ABB RobotStudio station: PiecePicking_20230616-110847.rsstn

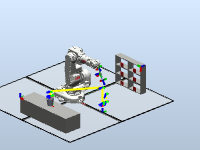
Station PiecePicking (saved by RobotStudio 6.8.8307.1040)
Controller System1
  mechanical unit ROB_1: IRB140_6_81_C_03, 6 joints, base frame (0, 0, 0) mm
Layout (positions relative to the parent item):
  - IRB140_6_81_C_03 [mechanism, from Robots\IRB140_6_81_C_G_03.rslib] at (0, 0, 0) mm; joint values [0, 0, 0, 0, 0.5236, 0] (rad or m)
  - Banda [part, from Libraries\Banda.rslib] at (-200, -850, 0) mm, rotated rx 90 ry 0 rz 90 deg
  - Balde [part, from Libraries\Balde.rslib] at (275, -710, 235) mm, rotated rx 90 ry 0 rz 90 deg
  - EstanteriaA  [part, from Libraries\EstanteriaA .rslib] at (0, 900, 0) mm, rotated rx 90 ry 0 rz 0 deg
  - Positioner_Balde [smart component, from Components\Positioner.rslib]
      properties: Object=Balde; Position=[0.275 -0.71 0.235]; Orientation=[1.5707963267949 0 1.5707963267949]; Reference=Global; ReferenceObject=(none)
  - Attacher_Balde [smart component, from Components\Attacher.rslib]
      properties: Parent=PF_Robotica; Flange=0; Child=Balde; Mount=false; Offset=[0 0 0]; Orientation=[0 0 0]
  - Detacher_Balde [smart component, from Components\Detacher.rslib]
      properties: Child=Balde; KeepPosition=true
  - PF_Robotica [mechanism, from Libraries\PF_Robotica.rslib] at (506.29, 0, 679.5) mm, rotated rx 180 ry 60 rz 180 deg
  - Pieza1 [smart component, from Libraries\Pieza1.rslib] at (-245.55, 1050.01, 0) mm
      connections:
        Pieza1.Pos_Pieza1 -> Positioner.Execute
        Pieza1.Attach_Pieza -> Attacher.Execute
        Pieza1.Detach_pieza -> Detacher.Execute
    - Positioner [smart component, from Components\Positioner.rslib] at (88.58, 803, 328) mm, rotated rx -90 ry 0 rz 0 deg
        properties: Object=PiezaTest_1; Position=[0.39675 0.803 0.328]; Orientation=[-1.5707963267949 0 0]; Reference=Global; ReferenceObject=(none)
    - PiezaTest_1 [part, from Libraries\Pieza1.rslib] at (642.3, -247.01, 328) mm, rotated rx -90 ry 0 rz 0 deg
    - Attacher [smart component, from Components\Attacher.rslib]
        properties: Parent=PF_Robotica; Flange=1; Child=PiezaTest_1; Mount=false; Offset=[0 0 0]; Orientation=[0 0 0]
    - Detacher [smart component, from Components\Detacher.rslib]
        properties: Child=PiezaTest_1; KeepPosition=true
  - Pieza2 [smart component, from Libraries\Pieza1.rslib] at (-251.26, 1022.75, 0) mm
      connections:
        Pieza2.Pos_Pieza1 -> Positioner.Execute
        Pieza2.Attach_Pieza -> Attacher.Execute
        Pieza2.Detach_pieza -> Detacher.Execute
    - Positioner [smart component, from Components\Positioner.rslib] at (88.58, 803, 328) mm, rotated rx -90 ry 0 rz 0 deg
        properties: Object=PiezaTest_1; Position=[0.13625 0.803 0.328]; Orientation=[-1.5707963267949 0 0]; Reference=Global; ReferenceObject=(none)
    - PiezaTest_1 [part, from Libraries\Pieza1.rslib] at (387.51, -219.75, 328) mm, rotated rx -90 ry 0 rz 0 deg
    - Attacher [smart component, from Components\Attacher.rslib]
        properties: Parent=PF_Robotica; Flange=1; Child=PiezaTest_1; Mount=false; Offset=[0 0 0]; Orientation=[0 0 0]
    - Detacher [smart component, from Components\Detacher.rslib]
        properties: Child=PiezaTest_1; KeepPosition=true
  - Pieza3 [smart component, from Libraries\Pieza1.rslib] at (-251.26, 1022.75, 0) mm
      connections:
        Pieza3.Pos_Pieza1 -> Positioner.Execute
        Pieza3.Attach_Pieza -> Attacher.Execute
        Pieza3.Detach_pieza -> Detacher.Execute
    - Positioner [smart component, from Components\Positioner.rslib] at (88.58, 803, 328) mm, rotated rx -90 ry 0 rz 0 deg
        properties: Object=PiezaTest_1; Position=[0.13625 0.803 0.189]; Orientation=[-1.5707963267949 0 0]; Reference=Global; ReferenceObject=(none)
    - PiezaTest_1 [part, from Libraries\Pieza1.rslib] at (387.51, -219.75, 189) mm, rotated rx -90 ry 0 rz 0 deg
    - Attacher [smart component, from Components\Attacher.rslib]
        properties: Parent=PF_Robotica; Flange=1; Child=PiezaTest_1; Mount=false; Offset=[0 0 0]; Orientation=[0 0 0]
    - Detacher [smart component, from Components\Detacher.rslib]
        properties: Child=PiezaTest_1; KeepPosition=true
  - Pieza4 [smart component, from Libraries\Pieza1.rslib] at (-251.26, 1022.75, 0) mm
      connections:
        Pieza4.Pos_Pieza1 -> Positioner.Execute
        Pieza4.Attach_Pieza -> Attacher.Execute
        Pieza4.Detach_pieza -> Detacher.Execute
    - Positioner [smart component, from Components\Positioner.rslib] at (88.58, 803, 328) mm, rotated rx -90 ry 0 rz 0 deg
        properties: Object=PiezaTest_1; Position=[0.39675 0.803 0.189]; Orientation=[-1.5707963267949 0 0]; Reference=Global; ReferenceObject=(none)
    - PiezaTest_1 [part, from Libraries\Pieza1.rslib] at (648.01, -219.75, 189) mm, rotated rx -90 ry 0 rz 0 deg
    - Attacher [smart component, from Components\Attacher.rslib]
        properties: Parent=PF_Robotica; Flange=1; Child=PiezaTest_1; Mount=false; Offset=[0 0 0]; Orientation=[0 0 0]
    - Detacher [smart component, from Components\Detacher.rslib]
        properties: Child=PiezaTest_1; KeepPosition=true
  - Pieza5 [smart component, from Libraries\Pieza1.rslib] at (-251.26, 1022.75, 0) mm
      connections:
        Pieza5.Pos_Pieza1 -> Positioner.Execute
        Pieza5.Attach_Pieza -> Attacher.Execute
        Pieza5.Detach_pieza -> Detacher.Execute
    - Positioner [smart component, from Components\Positioner.rslib] at (88.58, 803, 328) mm, rotated rx -90 ry 0 rz 0 deg
        properties: Object=PiezaTest_1; Position=[0.13625 0.803 0.042]; Orientation=[-1.5707963267949 0 0]; Reference=Global; ReferenceObject=(none)
    - PiezaTest_1 [part, from Libraries\Pieza1.rslib] at (387.51, -219.75, 42) mm, rotated rx -90 ry 0 rz 0 deg
    - Attacher [smart component, from Components\Attacher.rslib]
        properties: Parent=PF_Robotica; Flange=1; Child=PiezaTest_1; Mount=false; Offset=[0 0 0]; Orientation=[0 0 0]
    - Detacher [smart component, from Components\Detacher.rslib]
        properties: Child=PiezaTest_1; KeepPosition=true
  - Pieza6 [smart component, from Libraries\Pieza1.rslib] at (-251.26, 1022.75, 0) mm
      connections:
        Pieza6.Pos_Pieza1 -> Positioner.Execute
        Pieza6.Attach_Pieza -> Attacher.Execute
        Pieza6.Detach_pieza -> Detacher.Execute
    - Positioner [smart component, from Components\Positioner.rslib] at (88.58, 803, 328) mm, rotated rx -90 ry 0 rz 0 deg
        properties: Object=PiezaTest_1; Position=[0.39675 0.803 0.042]; Orientation=[-1.5707963267949 0 0]; Reference=Global; ReferenceObject=(none)
    - PiezaTest_1 [part, from Libraries\Pieza1.rslib] at (648.01, -219.75, 42) mm, rotated rx -90 ry 0 rz 0 deg
    - Attacher [smart component, from Components\Attacher.rslib]
        properties: Parent=PF_Robotica; Flange=1; Child=PiezaTest_1; Mount=false; Offset=[0 0 0]; Orientation=[0 0 0]
    - Detacher [smart component, from Components\Detacher.rslib]
        properties: Child=PiezaTest_1; KeepPosition=true
Attachment: PF_Robotica is attached to IRB140_6_81_C_03 / Link6
Attachment: Workobject_Est is attached to EstanteriaA 
Attachment: Workobject_1 is attached to Banda
Station signals: DI Balde_positioner, DI Pos_Pieza1, DI Pos_Pieza2, DI Pos_Pieza3, DI Pos_Pieza4, DI Pos_Pieza5, DI Pos_Pieza6, DI Pos_Piezas, DO DO_01, DO DO_02
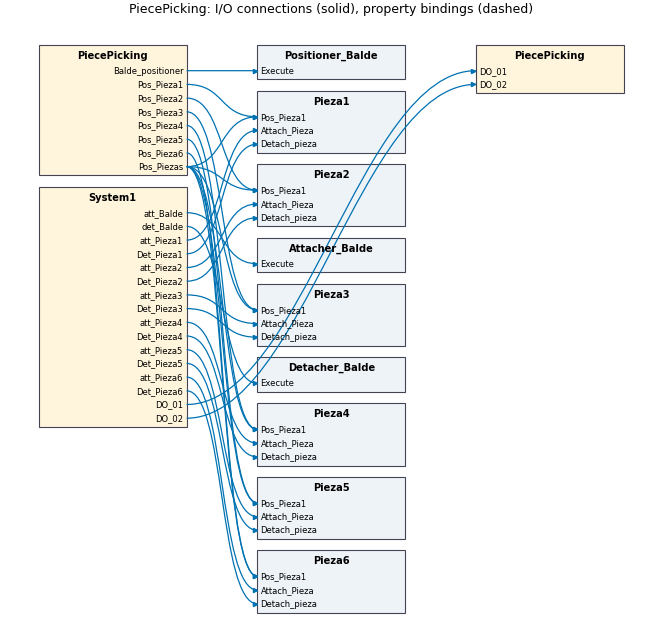
Station logic (signal -> signal, property => property):
  PiecePicking.Balde_positioner -> Positioner_Balde.Execute
  System1.att_Balde -> Attacher_Balde.Execute
  System1.det_Balde -> Detacher_Balde.Execute
  PiecePicking.Pos_Pieza1 -> Pieza1.Pos_Pieza1
  PiecePicking.Pos_Pieza2 -> Pieza2.Pos_Pieza1
  System1.att_Pieza1 -> Pieza1.Attach_Pieza
  System1.Det_Pieza1 -> Pieza1.Detach_pieza
  System1.att_Pieza2 -> Pieza2.Attach_Pieza
  System1.Det_Pieza2 -> Pieza2.Detach_pieza
  PiecePicking.Pos_Pieza3 -> Pieza3.Pos_Pieza1
  PiecePicking.Pos_Pieza4 -> Pieza4.Pos_Pieza1
  PiecePicking.Pos_Pieza5 -> Pieza5.Pos_Pieza1
  PiecePicking.Pos_Pieza6 -> Pieza6.Pos_Pieza1
  PiecePicking.Pos_Piezas -> Pieza6.Pos_Pieza1
  PiecePicking.Pos_Piezas -> Pieza5.Pos_Pieza1
  PiecePicking.Pos_Piezas -> Pieza4.Pos_Pieza1
  PiecePicking.Pos_Piezas -> Pieza3.Pos_Pieza1
  PiecePicking.Pos_Piezas -> Pieza2.Pos_Pieza1
  PiecePicking.Pos_Piezas -> Pieza1.Pos_Pieza1
  System1.att_Pieza3 -> Pieza3.Attach_Pieza
  System1.Det_Pieza3 -> Pieza3.Detach_pieza
  System1.att_Pieza4 -> Pieza4.Attach_Pieza
  System1.Det_Pieza4 -> Pieza4.Detach_pieza
  System1.att_Pieza5 -> Pieza5.Attach_Pieza
  System1.Det_Pieza5 -> Pieza5.Detach_pieza
  System1.att_Pieza6 -> Pieza6.Attach_Pieza
  System1.Det_Pieza6 -> Pieza6.Detach_pieza
  System1.DO_01 -> PiecePicking.DO_01
  System1.DO_02 -> PiecePicking.DO_02
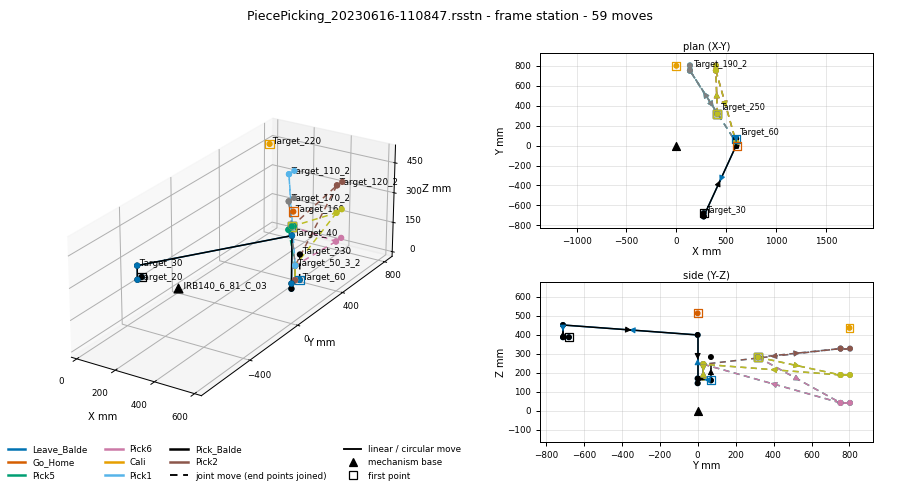
[picture p0: tool path of PiecePicking_20230616-110847.rsstn in frame station, 59 of 59 moves have a stored position in this frame; points joined in program order, loops and branches not executed]
Targets, tools, work objects and paths stored in the station, written as RAPID:
! task T_ROB1
MODULE CalibData
  TASK PERS wobjdata Workobject_1:=[FALSE,TRUE,"",[[-200,-850,230],[1,0,0,0]],[[475,140,0],[1,0,0,0]]];
  PERS tooldata TD_Hook:=[TRUE,[[68.38,0,60],[0.707106781,0.707106781,0,0]],[0.2,[28.798,-0.092,56.062],[1,0,0,0],0,0,0]];
  PERS tooldata TD_SuctionPad:=[TRUE,[[93.75,0,168.37],[0.970295726,0,0.241921896,0]],[0.2,[28.798,-0.092,56.062],[1,0,0,0],0,0,0]];
  TASK PERS wobjdata Workobject_Balde_Piso:=[FALSE,TRUE,"",[[600,0,0],[1,0,0,0]],[[0,0,0],[1,0,0,0]]];
  TASK PERS wobjdata Workobject_Est:=[FALSE,TRUE,"",[[533,800,437],[0.5,-0.5,0.5,0.5]],[[0,0,0],[1,0,0,0]]];
ENDMODULE

! task T_ROB1
MODULE Module1
  CONST robtarget Target_20:=[[-0.54180672,0.235098408,157.927793799],[0.499363871,0.499363893,0.500635292,-0.500635328],[-1,1,-2,0],[9E+09,9E+09,9E+09,9E+09,9E+09,9E+09]];
  CONST robtarget Target_10:=[[-0.541791285,31.542690631,157.927772118],[0.338220375,0.61994805,0.62152642,-0.339081557],[-1,1,-1,0],[9E+09,9E+09,9E+09,9E+09,9E+09,9E+09]];
  CONST robtarget Target_30:=[[-0.541814528,0.23509908,222.389598203],[0.499363884,0.49936382,0.500635317,-0.500635363],[-1,1,-2,0],[9E+09,9E+09,9E+09,9E+09,9E+09,9E+09]];
  CONST robtarget Target_40:=[[0,0,400],[0.499363884,0.49936382,0.500635317,-0.500635363],[0,1,-3,0],[9E+09,9E+09,9E+09,9E+09,9E+09,9E+09]];
  CONST robtarget Target_50:=[[-0.038127492,-0.000030739,145.519742619],[0.499363836,0.499363825,0.500635306,-0.500635416],[-1,2,-3,0],[9E+09,9E+09,9E+09,9E+09,9E+09,9E+09]];
  CONST robtarget Target_60:=[[0,70,160.52],[0.182019153,0.682470244,0.683552682,-0.184008491],[0,2,-2,0],[9E+09,9E+09,9E+09,9E+09,9E+09,9E+09]];
  CONST robtarget Target_80:=[[-77.125218661,-72.22939491,-596.502903487],[0.618449548,0.618449544,0.342812142,0.342812128],[0,-1,0,0],[9E+09,9E+09,9E+09,9E+09,9E+09,9E+09]];
  CONST robtarget Target_90:=[[204.199229947,-72.229383295,-619.023797732],[0.618449546,0.618449531,0.34281213,0.342812167],[0,-2,1,0],[9E+09,9E+09,9E+09,9E+09,9E+09,9E+09]];
  CONST robtarget Target_50_2:=[[-0.038127492,-0.000030739,170.519742619],[0.182018295,0.682471059,0.683552878,-0.184005593],[-1,1,-2,0],[9E+09,9E+09,9E+09,9E+09,9E+09,9E+09]];
  CONST robtarget Target_110:=[[109,396.75,3],[1,0,0,0],[0,2,-2,0],[9E+09,9E+09,9E+09,9E+09,9E+09,9E+09]];
  CONST robtarget Target_120:=[[109,136.25,3],[1,0,0,0],[0,1,-2,0],[9E+09,9E+09,9E+09,9E+09,9E+09,9E+09]];
  CONST robtarget Target_130:=[[108.313469676,92.052338402,147.49758099],[0.444719526,0.257906476,0.743119571,0.428348101],[0,-2,-2,0],[9E+09,9E+09,9E+09,9E+09,9E+09,9E+09]];
  CONST robtarget Target_50_3_2:=[[0.216181367,29.999981348,245.519415627],[0.611593294,0.353103544,0.613150552,-0.354002726],[0,-3,2,0],[9E+09,9E+09,9E+09,9E+09,9E+09,9E+09]];
  CONST robtarget Target_150:=[[0.216193734,29.999948387,175.359992959],[0.611593362,0.353103485,0.613150461,-0.354002825],[0,-2,1,0],[9E+09,9E+09,9E+09,9E+09,9E+09,9E+09]];
  CONST robtarget Target_110_2:=[[109,396.75,-47],[1,0,0,0],[0,2,-2,0],[9E+09,9E+09,9E+09,9E+09,9E+09,9E+09]];
  CONST robtarget Target_160:=[[605.229348481,0,514.125118395],[0.275637355,0,0.961261696,0],[0,0,0,0],[9E+09,9E+09,9E+09,9E+09,9E+09,9E+09]];
  CONST robtarget Target_170:=[[248,396.75,3],[0.216439613,0,0,0.976296007],[0,2,-2,0],[9E+09,9E+09,9E+09,9E+09,9E+09,9E+09]];
  CONST robtarget Target_180:=[[248,136.25,3],[0.707106781,0,0,0.707106781],[0,1,-2,0],[9E+09,9E+09,9E+09,9E+09,9E+09,9E+09]];
  CONST robtarget Target_190:=[[395,396.75,3],[0.382683432,0,0,0.923879533],[0,2,-2,0],[9E+09,9E+09,9E+09,9E+09,9E+09,9E+09]];
  CONST robtarget Target_200:=[[395,136.25,3],[0.707106781,0,0,0.707106781],[0,1,-2,0],[9E+09,9E+09,9E+09,9E+09,9E+09,9E+09]];
  CONST robtarget Target_120_2:=[[109,136.25,-47],[1,0,0,0],[0,1,-2,0],[9E+09,9E+09,9E+09,9E+09,9E+09,9E+09]];
  CONST robtarget Target_170_2:=[[248,396.75,-47],[0.216439613,0,0,0.976296007],[0,2,-2,0],[9E+09,9E+09,9E+09,9E+09,9E+09,9E+09]];
  CONST robtarget Target_180_2:=[[248,136.25,-47],[0.707106781,0,0,0.707106781],[0,1,-2,0],[9E+09,9E+09,9E+09,9E+09,9E+09,9E+09]];
  CONST robtarget Target_190_2:=[[395,396.75,-47],[0.382683432,0,0,0.923879533],[0,2,-2,0],[9E+09,9E+09,9E+09,9E+09,9E+09,9E+09]];
  CONST robtarget Target_200_2:=[[395,136.25,-47],[0.707106781,0,0,0.707106781],[0,1,-2,0],[9E+09,9E+09,9E+09,9E+09,9E+09,9E+09]];
  CONST robtarget Target_60_2:=[[0,70,280.52],[0.182019153,0.682470244,0.683552682,-0.184008491],[0,-2,-2,0],[9E+09,9E+09,9E+09,9E+09,9E+09,9E+09]];
  CONST robtarget Target_220:=[[0,533,0],[1,0,0,0],[1,2,2,0],[9E+09,9E+09,9E+09,9E+09,9E+09,9E+09]];
  CONST robtarget Target_230:=[[0.000068646,70.00001103,283.574285968],[0.182019117,0.682470266,0.683552671,-0.184008489],[0,2,-2,0],[9E+09,9E+09,9E+09,9E+09,9E+09,9E+09]];
  CONST robtarget Target_250:=[[-188.843410439,317.985657737,282.635376599],[0.28601825,0.002111346,-0.703849705,-0.650218959],[0,1,-1,0],[9E+09,9E+09,9E+09,9E+09,9E+09,9E+09]];
  PROC Main()
    Go_Home;
    Pick_Balde;
    Pick1;
    Pick2;
    Pick3;
    Leave_Balde;
    Go_Home;
  ENDPROC
  PROC Leave_Balde()
    MoveJ Target_60,vel,fine,TD_Hook\WObj:=Workobject_Balde_Piso;
    MoveJ Target_50_2,v50,z10,TD_Hook\WObj:=Workobject_Balde_Piso;
    MoveJ Target_50,v50,fine,TD_Hook\WObj:=Workobject_Balde_Piso;
    WaitTime 0.5;
    MoveL Target_40,vel,z150,TD_Hook\WObj:=Workobject_Balde_Piso;
    MoveL Target_30,vel,z100,TD_Hook\WObj:=Workobject_1;
    MoveL Target_20,v100,fine,TD_Hook\WObj:=Workobject_1;
    WaitTime 0.5;
    MoveL Target_10,vel,z100,TD_Hook\WObj:=Workobject_1;
  ENDPROC
  PROC Go_Home()
    MoveJ Target_160,vel,z0,TD_SuctionPad\WObj:=wobj0;
  ENDPROC
  PROC Pick5()
    MoveJ Target_250,vel,z5,TD_SuctionPad\WObj:=Workobject_Balde_Piso;
    MoveJ Target_190_2,vel,z5,TD_SuctionPad\WObj:=Workobject_Est;
    PulseDO DO_02;
    MoveL Target_190,v50,fine,TD_SuctionPad\WObj:=Workobject_Est;
    WaitTime 1;
    MoveL Target_190_2,v50,z10,TD_SuctionPad\WObj:=Workobject_Est;
    MoveJ Target_50_3_2,vel,z50,TD_SuctionPad\WObj:=Workobject_Balde_Piso;
    MoveL Target_150,v50,fine,TD_SuctionPad\WObj:=Workobject_Balde_Piso;
    PulseDO DO_01;
    WaitTime 1;
    MoveJ Target_50_3_2,vel,z50,TD_SuctionPad\WObj:=Workobject_Balde_Piso;
  ENDPROC
  PROC Pick6()
    MoveJ Target_250,vel,z5,TD_SuctionPad\WObj:=Workobject_Balde_Piso;
    MoveJ Target_200_2,vel,z5,TD_SuctionPad\WObj:=Workobject_Est;
    PulseDO DO_02;
    MoveL Target_200,v50,fine,TD_SuctionPad\WObj:=Workobject_Est;
    WaitTime 1;
    MoveL Target_200_2,v50,z10,TD_SuctionPad\WObj:=Workobject_Est;
    MoveJ Target_50_3_2,vel,z50,TD_SuctionPad\WObj:=Workobject_Balde_Piso;
    MoveL Target_150,v50,fine,TD_SuctionPad\WObj:=Workobject_Balde_Piso;
    PulseDO DO_01;
    WaitTime 1;
    MoveJ Target_50_3_2,vel,z50,TD_SuctionPad\WObj:=Workobject_Balde_Piso;
  ENDPROC
  PROC Cali()
    MoveJ Target_220,v200,z5,TD_SuctionPad\WObj:=Workobject_Est;
  ENDPROC
  PROC Pick1()
    MoveJ Target_250,vel,z5,TD_SuctionPad\WObj:=Workobject_Balde_Piso;
    MoveJ Target_110_2,vel,z5,TD_SuctionPad\WObj:=Workobject_Est;
    PulseDO DO_02;
    MoveL Target_110,v50,fine,TD_SuctionPad\WObj:=Workobject_Est;
    WaitTime 1;
    MoveL Target_110_2,vel,z100,TD_SuctionPad\WObj:=Workobject_Est;
    MoveJ Target_50_3_2,vel,z5,TD_SuctionPad\WObj:=Workobject_Balde_Piso;
    MoveL Target_150,vel,fine,TD_SuctionPad\WObj:=Workobject_Balde_Piso;
    PulseDO DO_01;
    WaitTime 1;
    MoveJ Target_50_3_2,vel,z5,TD_SuctionPad\WObj:=Workobject_Balde_Piso;
  ENDPROC
  PROC Pick_Balde()
    MoveJ Target_10,vel,z100,TD_Hook\WObj:=Workobject_1;
    MoveL Target_20,vel,fine,TD_Hook\WObj:=Workobject_1;
    WaitTime 0.5;
    MoveL Target_30,v200,z100,TD_Hook\WObj:=Workobject_1;
    MoveL Target_40,v200,fine,TD_Hook\WObj:=Workobject_Balde_Piso;
    WaitTime 1;
    MoveL Target_50,v200,fine,TD_Hook\WObj:=Workobject_Balde_Piso;
    WaitTime 0.5;
    MoveJ Target_50_2,v50,fine,TD_Hook\WObj:=Workobject_Balde_Piso;
    MoveJ Target_60,vel,z10,TD_Hook\WObj:=Workobject_Balde_Piso;
    MoveJ Target_230,vel,z5,TD_Hook\WObj:=Workobject_Balde_Piso;
  ENDPROC
  PROC Pick2()
    MoveJ Target_250,vel,z5,TD_SuctionPad\WObj:=Workobject_Balde_Piso;
    MoveJ Target_120_2,vel,z5,TD_SuctionPad\WObj:=Workobject_Est;
    PulseDO DO_02;
    MoveL Target_120,v50,fine,TD_SuctionPad\WObj:=Workobject_Est;
    WaitTime 1;
    MoveL Target_120_2,v50,z10,TD_SuctionPad\WObj:=Workobject_Est;
    MoveJ Target_50_3_2,vel,z50,TD_SuctionPad\WObj:=Workobject_Balde_Piso;
    MoveL Target_150,v50,fine,TD_SuctionPad\WObj:=Workobject_Balde_Piso;
    PulseDO DO_01;
    WaitTime 1;
    MoveJ Target_50_3_2,vel,z50,TD_SuctionPad\WObj:=Workobject_Balde_Piso;
  ENDPROC
  PROC Pick3()
    MoveJ Target_250,vel,z5,TD_SuctionPad\WObj:=Workobject_Balde_Piso;
    MoveJ Target_170_2,vel,z5,TD_SuctionPad\WObj:=Workobject_Est;
    PulseDO DO_02;
    MoveL Target_170,v50,fine,TD_SuctionPad\WObj:=Workobject_Est;
    WaitTime 1;
    MoveL Target_170_2,v50,z10,TD_SuctionPad\WObj:=Workobject_Est;
    MoveJ Target_50_3_2,vel,z50,TD_SuctionPad\WObj:=Workobject_Balde_Piso;
    MoveL Target_150,v50,fine,TD_SuctionPad\WObj:=Workobject_Balde_Piso;
    PulseDO DO_01;
    WaitTime 1;
    MoveJ Target_50_3_2,vel,z50,TD_SuctionPad\WObj:=Workobject_Balde_Piso;
  ENDPROC
  PROC Pick4()
    MoveJ Target_250,vel,z5,TD_SuctionPad\WObj:=Workobject_Balde_Piso;
    MoveJ Target_180_2,vel,z5,TD_SuctionPad\WObj:=Workobject_Est;
    PulseDO DO_02;
    MoveL Target_180,v50,fine,TD_SuctionPad\WObj:=Workobject_Est;
    WaitTime 1;
    MoveL Target_180_2,v50,z10,TD_SuctionPad\WObj:=Workobject_Est;
    MoveJ Target_50_3_2,vel,z50,TD_SuctionPad\WObj:=Workobject_Balde_Piso;
    MoveL Target_150,v50,fine,TD_SuctionPad\WObj:=Workobject_Balde_Piso;
    PulseDO DO_01;
    WaitTime 1;
    MoveJ Target_50_3_2,vel,z50,TD_SuctionPad\WObj:=Workobject_Balde_Piso;
  ENDPROC
ENDMODULE

